// TIA Portal V17 export
// export: Created 2024-06-16T17:47:34.8628858Z, ExportSetting WithDefaults, DisplayName Totally Integrated Automation Portal, DisplayVersion V17, DisplayName TIA Portal Openness, DisplayVersion V17, DisplayName TIA Portal Version Control Interface, DisplayVersion V17, DisplayName STEP 7 Professional, DisplayVersion V17, DisplayName STEP 7 Safety, DisplayVersion V17, DisplayName WinCC Professional, DisplayVersion V17
FUNCTION "G7A_St4" : Void   // FC405, LAD
{ S7_Optimized_Access := 'TRUE' }
VERSION : 0.1
// stored: AutoNumber false, IsIECCheckEnabled false, SetENOAutomatically false, UDAEnableTagReadback false
BEGIN

REGION Network 1: G7 Auto --> Station 4 : Marquage
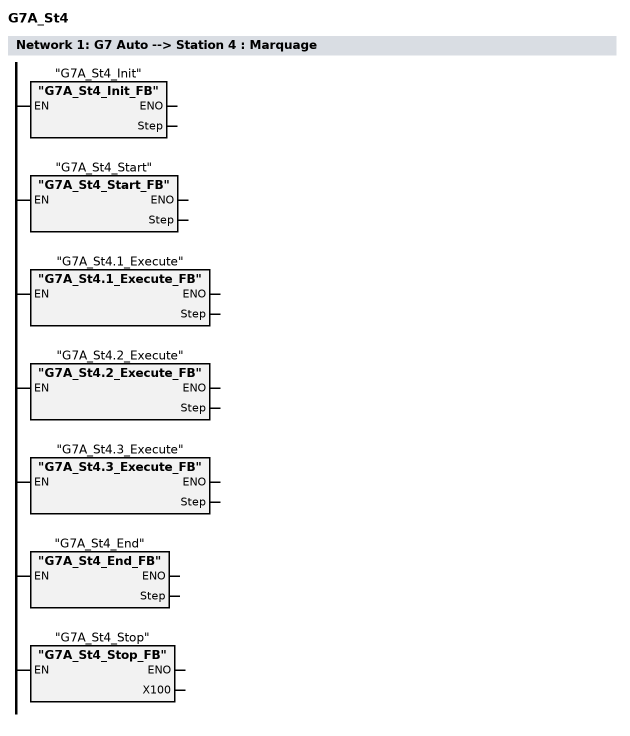
   RUNG wire#powerrail
      "G7A_St4_Init"("Step" =>)
   END_RUNG
   RUNG wire#powerrail
      "G7A_St4_Start"("Step" =>)
   END_RUNG
   RUNG wire#powerrail
      "G7A_St4.1_Execute"("Step" =>)
   END_RUNG
   RUNG wire#powerrail
      "G7A_St4.2_Execute"("Step" =>)
   END_RUNG
   RUNG wire#powerrail
      "G7A_St4.3_Execute"("Step" =>)
   END_RUNG
   RUNG wire#powerrail
      "G7A_St4_End"("Step" =>)
   END_RUNG
   RUNG wire#powerrail
      "G7A_St4_Stop"(X100 =>)
   END_RUNG
   // the same network as SCL:
   "G7A_St4_Init"();   // "G7A_St4_Init_FB"
   "G7A_St4_Start"();   // "G7A_St4_Start_FB"
   "G7A_St4.1_Execute"();   // "G7A_St4.1_Execute_FB"
   "G7A_St4.2_Execute"();   // "G7A_St4.2_Execute_FB"
   "G7A_St4.3_Execute"();   // "G7A_St4.3_Execute_FB"
   "G7A_St4_End"();   // "G7A_St4_End_FB"
   "G7A_St4_Stop"();   // "G7A_St4_Stop_FB"
END_REGION
END_FUNCTION
